Yaskawa INFORM job: white_plate_planes_program.JBI

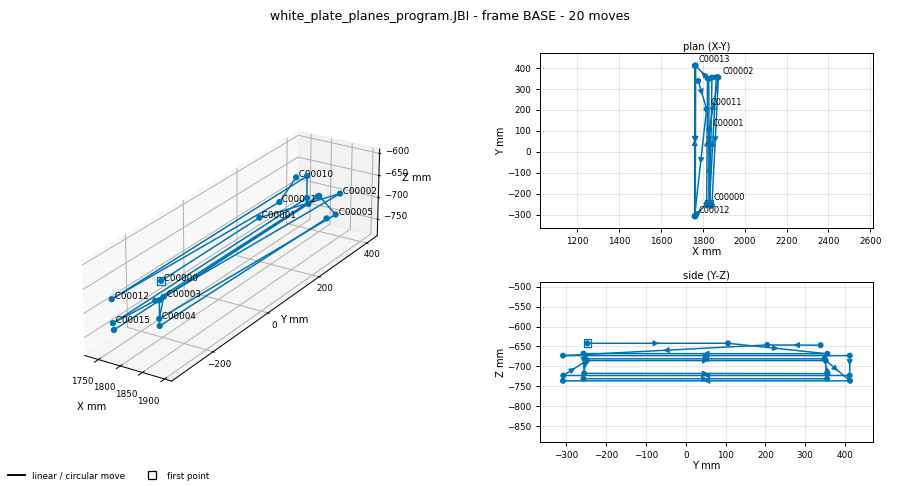
[picture p0: tool path of white_plate_planes_program.JBI in frame BASE, 20 of 23 moves have a stored position in this frame; points joined in program order, loops and branches not executed]
/JOB
//NAME white_plate_planes_program
//POS
///NPOS 20,0,20,0,0,0
///TOOL 0
///POSTYPE BASE
///RECTAN
///RCONF 0,0,0,0,0,0,0,0,0,0,0,0,0,0,0,0,0,0,0,0,0,0,0,0
C00000=1830.802427,-246.862154,-641.935850,175.000000,-89.101197,-5.000000
C00001=1830.059198,106.088885,-641.936847,175.000000,-89.101197,-5.000000
C00002=1873.896110,355.497164,-668.253070,175.000000,-89.101197,-5.000000
C00003=1842.888754,-257.052128,-667.744668,175.000000,-89.101197,-5.000000
C00004=1830.768242,-255.212026,-717.560742,175.000000,-89.101197,-5.000000
C00005=1863.784244,356.187016,-718.100614,175.000000,-89.101197,-5.000000
C00006=1828.086394,348.126364,-680.943915,175.000000,-89.101197,-5.000000
C00007=1828.853319,-251.546408,-680.934444,175.000000,-89.101197,-5.000000
C00008=1832.894122,-257.303711,-731.003782,175.000000,-89.101197,-5.000000
C00009=1843.051373,354.883523,-731.185078,180.000000,-60.000000,0.000000
C00010=1777.408261,338.617857,-646.732027,5.000000,-89.091122,175.000000
C00011=1817.446172,204.524658,-646.098030,5.000000,-89.091122,175.000000
C00012=1760.049958,-308.440896,-672.944436,5.000000,-89.091122,175.000000
C00013=1761.203328,411.893863,-672.919740,5.000000,-89.091122,175.000000
C00014=1761.864353,411.663340,-722.915547,5.000000,-89.091122,175.000000
C00015=1760.883365,-307.665195,-722.937499,5.000000,-89.091122,175.000000
C00016=1817.839207,-248.630374,-685.437139,5.000000,-89.091122,175.000000
C00017=1821.803484,351.637717,-685.368916,5.000000,-89.091122,175.000000
C00018=1765.103107,412.575313,-736.274201,5.000000,-89.091122,175.000000
C00019=1763.377310,-308.350147,-736.307982,180.000000,-60.000000,0.000000
///POSTYPE PULSE
///PULSE
EC00000=0.0
EC00001=0.0
EC00002=0.0
EC00003=0.0
EC00004=0.0
EC00005=0.0
EC00006=0.0
EC00007=0.0
EC00008=0.0
EC00009=0.0
EC00010=184320.0
EC00011=184320.0
EC00012=184320.0
EC00013=184320.0
EC00014=184320.0
EC00015=184320.0
EC00016=184320.0
EC00017=184320.0
EC00018=184320.0
EC00019=184320.0
//INST
///DATE 2023/08/16 18:09
///ATTR SC,RW,RJ
////FRAME BASE
///GROUP1 RB1,ST1
NOP
MOVJ P009 EX000 VJ=15.00
MOVJ C00000 EC00000 VJ=15.0
CALL JOB:SPYON
MOVL C00001 EC00001 V=150.0
MOVL C00002 EC00002 V=150.0
MOVL C00003 EC00003 V=150.0
MOVL C00004 EC00004 V=150.0
MOVL C00005 EC00005 V=150.0
MOVL C00006 EC00006 V=150.0
MOVL C00007 EC00007 V=150.0
MOVL C00008 EC00008 V=150.0
MOVL C00009 EC00009 V=150.0
CALL JOB:SPYOF
MOVJ P009 VJ=15.00
MOVJ C00010 EC00010 VJ=15.0
CALL JOB:SPYON
MOVL C00011 EC00011 V=150.0
MOVL C00012 EC00012 V=150.0
MOVL C00013 EC00013 V=150.0
MOVL C00014 EC00014 V=150.0
MOVL C00015 EC00015 V=150.0
MOVL C00016 EC00016 V=150.0
MOVL C00017 EC00017 V=150.0
MOVL C00018 EC00018 V=150.0
MOVL C00019 EC00019 V=150.0
CALL JOB:SPYOF
MOVJ P009 VJ=15.00
END
